Universal Robots PolyScope program: Main.urp

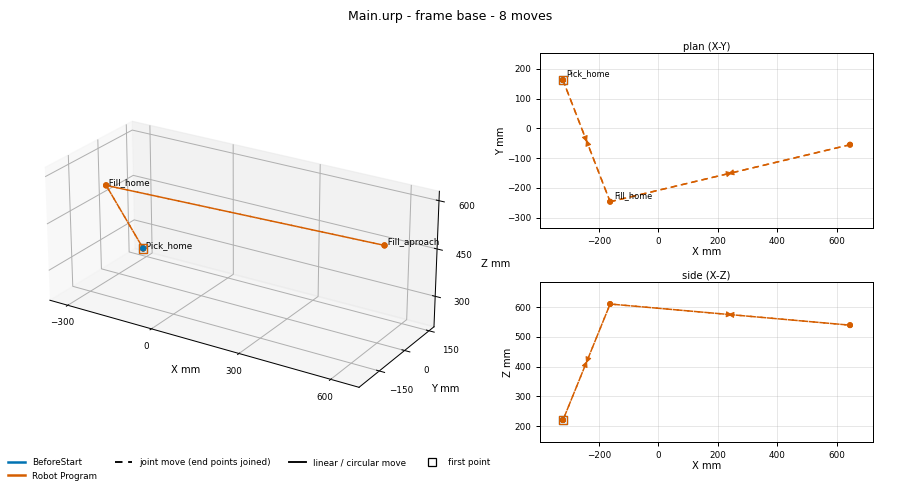
[picture p0: tool path of Main.urp in frame base, 8 of 9 moves have a stored position in this frame; points joined in program order, loops and branches not executed]
Program Main (installation=default directory=/programs/RegalRexnord createdIn=3.12.1.90940 lastSavedIn=3.12.1.90940 robotSerialNumber=2016301828)
Calibrated DH parameters: a=[-0.000087, -0.6088, -0.564866, 0.000367, -0.00029, 0]; d=[0.127939, 20.625424, -41.590771, 21.128581, 0.115471, 0.092056]; alpha=[1.57116, -0.003242, -0.004054, 1.570309, -1.570517, 0]; deltaTheta=[-0.000043, -0.109409, 0.258819, -0.149504, -0.000092, 0.000021]
InitVariablesNode variables(variable(name=Rack_number, expression=2), variable(name=Row_full, expression=True), variable(name=Row_number, expression=9), variable(name=Var_point, expression=Point_1), variable(name=i, expression=1), variable(name=ir_value, expression=False), variable(name=j, expression=1), variable(name=tcpforces, expression=get_tcp_force()), variable(name=torqueX, expression=0), variable(name=torqueY, expression=0))
BeforeStart
  SuppressedNode
    First_point_ := p[0.10705,0.15735,0.05121,0.028,3.109,0.517]
  SuppressedNode
    Var_point := pose_add(First_point_, p[0,0.03289,0.01197,0,0,0])
  Set DigitalOutput pin=digital_out[0]; digitalValue=0
  Set DigitalOutput pin=digital_out[1]; digitalValue=0
  pose1 := pose_add(Point_1, p[0.01197,0,0.03289,0,0,0])
  pose2 := pose_add(Point_2, p[0.01197,0,0.03289,0,0,0])
  pose3 := pose_add(Point_3, p[0.01197,0,0.03289,0,0,0])
  pose4 := pose_add(Point_4, p[0.01197,0,0.03289,0,0,0])
  pose5 := pose_add(Point_5, p[0.01197,0,0.03289,0,0,0])
  pose6 := pose_add(Point_6, p[0.01197,0,0.03289,0,0,0])
  pose7 := pose_add(Point_7, p[0.01197,0,0.03289,0,0,0])
  pose8 := pose_add(Point_8, p[0.01197,0,0.03289,0,0,0])
  pose9 := pose_add(Point_9, p[0.01197,0,0.03289,0,0,0])
  poses := [pose1,pose2,pose3,pose4,pose5,pose6,pose7,pose8,pose9]
  pose10 := pose_add(Point_10, p[0.01197,0,0.03289,0,0,0])
  pose11 := pose_add(Point_11, p[0.01197,0,0.03289,0,0,0])
  pose12 := pose_add(Point_12, p[0.01197,0,0.03289,0,0,0])
  pose13 := pose_add(Point_13, p[0.01197,0,0.03289,0,0,0])
  pose14 := pose_add(Point_14, p[0.01197,0,0.03289,0,0,0])
  pose15 := pose_add(Point_15, p[0.01197,0,0.03289,0,0,0])
  pose16 := pose_add(Point_16, p[0.01197,0,0.03289,0,0,0])
  pose17 := pose_add(Point_17, p[0.01197,0,0.03289,0,0,0])
  pose18 := pose_add(Point_18, p[0.01197,0,0.03289,0,0,0])
  poses2 := [pose10,pose11,pose12,pose13,pose14,pose15,pose16,pose17,pose18]
  Var_point := pose10
  MoveJ speed 120 deg/s, acceleration 120 deg/s^2 (useActiveTCP=true)
    Waypoint Pick_home: TCP in base x=-320.57 y=162.039 z=220.257 mm, rx=1.2082 ry=-1.21 rz=-1.2062 rad; joints [-180, -70, -150, -140.003, 269.997, -0.001] deg; flange x=-320.609 y=162.049 z=220.3 mm, rx=1.2082 ry=-1.2099 rz=-1.2063 rad
Robot Program (runOnlyOnce=true)
  Loop While (checkContinuously=false) expression=i≤Rack_number
    Loop While (checkContinuously=false) expression=j≤Row_number
      Folder Assign point
        If i==1
          Var_point := poses[j-1]
        ElseIf i==2
          Var_point := poses2[j-1]
      Loop While (checkContinuously=false) expression=Row_full== True
        Folder Pick & place sequence
          MoveL speed 1000 mm/s, acceleration 1500 mm/s^2 (useActiveTCP=true) feature=Base
            Waypoint Waypoint (Variable): variable=Var_point
          Wait Sleep waitTime=0.25
          Folder Check sensor
            If ir_value== True
              Row_full := True
            Else 
              Row_full := False
          If Row_full== True
            MoveL speed 20 mm/s, acceleration 1500 mm/s^2 (useActiveTCP=true) feature=Joint_6_name
              MoveDirectionNode (selectedDirection=YMinus toolParams=0.05, 1.5) feature=Joint_6_name
                Until DISTANCE (allowActions=false deceleration=3 distanceNodeType=STOP) Distance=0.035; motionParameters(blendRadius=0)
              Set DigitalOutput pin=digital_out[0]; digitalValue=1
              Set NoAction (payload=1.5 tcpAsCog=true)
              Wait Sleep waitTime=0.25
              MoveDirectionNode (selectedDirection=YPlus) feature=Joint_6_name
                Until DISTANCE (allowActions=false deceleration=3 distanceNodeType=BLEND) Distance=0.005; motionParameters(blendRadius=0)
              Set DigitalOutput pin=digital_out[1]; digitalValue=1
              MoveDirectionNode (selectedDirection=YPlus) feature=Joint_6_name
                Until DISTANCE (allowActions=false deceleration=3 distanceNodeType=STOP) Distance=0.031; motionParameters(blendRadius=0)
              Wait Sleep waitTime=0.25
              MoveDirectionNode (selectedDirection=ZMinus toolParams=0.03, 1.5) feature=Joint_6_name
                Until DISTANCE (allowActions=false deceleration=3 distanceNodeType=BLEND) Distance=0.08; motionParameters(blendRadius=0.02)
            If 4<j
              MoveL speed 800 mm/s, acceleration 2000 mm/s^2 (useActiveTCP=true) feature=Base
                Waypoint Pick_home: motionParameters(blendRadius=0.087); TCP in base x=-320.57 y=162.039 z=220.257 mm, rx=1.2082 ry=-1.21 rz=-1.2062 rad; joints [-180, -70, -150, -140.003, 269.997, -0.001] deg; flange x=-320.609 y=162.049 z=220.3 mm, rx=1.2082 ry=-1.2099 rz=-1.2063 rad
            MoveJ speed 180 deg/s, acceleration 240 deg/s^2 (useActiveTCP=true)
              Waypoint Fill_home: motionParameters(blendRadius=0.4); TCP in base x=-162.031 y=-246.748 z=610.546 mm, rx=-3.1414 ry=-0.0066 rz=-0.0059 rad; joints [-90.002, -69.999, -110, -270, 269.997, -0.004] deg; flange x=-162.029 y=-246.755 z=610.494 mm, rx=-3.1412 ry=-0.0066 rz=-0.0059 rad
              Waypoint Fill_aproach: TCP in base x=644.574 y=-55.044 z=539.475 mm, rx=-2.2175 ry=-2.2214 rz=-0.0032 rad; joints [9.62, -106.707, -81.523, -261.754, 270.133, 9.714] deg; flange x=644.592 y=-55.009 z=539.434 mm, rx=-2.2174 ry=-2.2214 rz=-0.003 rad
              SuppressedNode
                Set DigitalOutput pin=digital_out[1]; digitalValue=0
              Wait Sleep waitTime=1
            MoveL speed 30 mm/s, acceleration 500 mm/s^2 (useActiveTCP=true) feature=Base
              MoveDirectionNode (selectedDirection=ZMinus)
                Until DISTANCE (allowActions=false deceleration=3 distanceNodeType=STOP) Distance=0.195; motionParameters(blendRadius=0)
                Until EXPRESSION (allowActions=false) ExpressionBranch=2.5<torqueY
            MoveL speed 250 mm/s, acceleration 1500 mm/s^2 (useActiveTCP=true) feature=Base
              MoveDirectionNode (selectedDirection=ZPlus)
                Until DISTANCE (allowActions=false deceleration=3 distanceNodeType=BLEND) Distance=0.01; motionParameters(blendRadius=0)
              Set DigitalOutput pin=digital_out[1]; digitalValue=0
              Wait Sleep waitTime=0.5
              Set DigitalOutput pin=digital_out[0]; digitalValue=0
              Set NoAction (payload=0.6 tcpAsCog=true)
            MoveL speed 500 mm/s, acceleration 1500 mm/s^2 (useActiveTCP=true) feature=Base
              Waypoint Filling_aproach: TCP in base x=644.567 y=-55.04 z=539.506 mm, rx=-2.2175 ry=-2.2215 rz=-0.0033 rad; joints [9.62, -106.707, -81.523, -261.754, 270.133, 9.714] deg; flange x=644.592 y=-55.009 z=539.434 mm, rx=-2.2174 ry=-2.2214 rz=-0.003 rad
            MoveJ speed 180 deg/s, acceleration 180 deg/s^2 (useActiveTCP=true)
              Waypoint Fill_home: motionParameters(blendRadius=0.5); TCP in base x=-162.031 y=-246.748 z=610.546 mm, rx=-3.1414 ry=-0.0066 rz=-0.0059 rad; joints [-90.002, -69.999, -110, -270, 269.997, -0.004] deg; flange x=-162.029 y=-246.755 z=610.494 mm, rx=-3.1412 ry=-0.0066 rz=-0.0059 rad
            MoveJ speed 120 deg/s, acceleration 160 deg/s^2 (useActiveTCP=true)
              Waypoint Pick_home: motionParameters(jointSpeed=2.792527 jointAcceleration=3.490659 cartesianSpeed=0.25 cartesianAcceleration=1.2); TCP in base x=-320.57 y=162.039 z=220.257 mm, rx=1.2082 ry=-1.21 rz=-1.2062 rad; joints [-180, -70, -150, -140.003, 269.997, -0.001] deg; flange x=-320.609 y=162.049 z=220.3 mm, rx=1.2082 ry=-1.2099 rz=-1.2063 rad
          Else 
            MoveL speed 250 mm/s, acceleration 1200 mm/s^2 (useActiveTCP=true) feature=Joint_6_name
              MoveDirectionNode (selectedDirection=ZMinus)
                Until DISTANCE (allowActions=false deceleration=3 distanceNodeType=BLEND) Distance=0.07; motionParameters(blendRadius=0.02)
              MoveDirectionNode (selectedDirection=XMinus)
                Until DISTANCE (allowActions=false deceleration=3 distanceNodeType=STOP) Distance=0.125; motionParameters(blendRadius=0)
      SuppressedNode
        Var_point := pose_trans(Var_point, p[-Row_dist,0,0,0,0,0])
      j := j+1
      Row_full := True
    j := 1
    MoveL speed 1000 mm/s, acceleration 1500 mm/s^2 (useActiveTCP=true) feature=Base
      Waypoint Pick_home: TCP in base x=-320.57 y=162.039 z=220.257 mm, rx=1.2082 ry=-1.21 rz=-1.2062 rad; joints [-180, -70, -150, -140.003, 269.997, -0.001] deg; flange x=-320.609 y=162.049 z=220.3 mm, rx=1.2082 ry=-1.2099 rz=-1.2063 rad
    SuppressedNode
      Var_point := pose_add(First_point_, p[0,Rack_distY*i,0,0,0,0])
    i := i+1
  Halt
Thread Thread_1 (runOnlyOnce=false)
  Wait Sleep waitTime=0.01
  tcpforces := get_tcp_force()
  torqueY := tcpforces[4]
  torqueX := tcpforces[3]
Thread Thread_2 (runOnlyOnce=false)
  Wait Sleep waitTime=0.01
  ir_value := digital_in[1]
